INTERFACE I_TraceLogger

METHOD LogMessage
VAR_INPUT
	Key		  : T_MaxString;
	Value	  : T_MaxString;
	SourceId  : UDINT := 0;
	TimeStamp : ULINT := 0;
	MessageId : UDINT := 1;
	Severity  : USINT := 1;
END_VAR
END_METHOD

END_INTERFACE

(* stored: Version 1.1.0.1
   Itf I_TraceLogger: Id {65a75728-6630-458f-a11a-131852730d4e}
   Method LogMessage: Id {bc47b5b5-7e08-47ae-8fbd-08e46e2940aa} *)
